// TIA Portal V18 export
FUNCTION "TCS" : Void   // FC3, LAD
{ S7_Optimized_Access := 'TRUE' }
VERSION : 0.1
// stored: AutoNumber true, IsIECCheckEnabled false, SetENOAutomatically false, UDAEnableTagReadback false
BEGIN

REGION Network 1
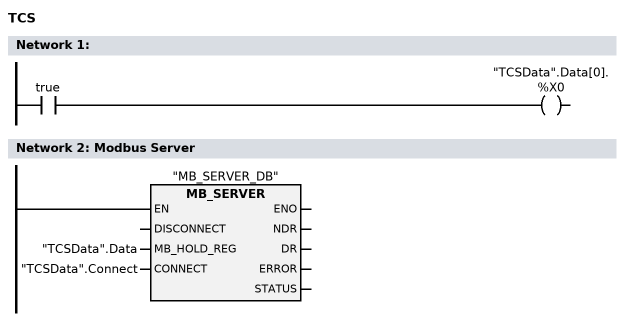
   RUNG wire#powerrail
      Contact( true )
      Coil( "TCSData".Data[0].%X0 )
   END_RUNG
   // the same network as SCL:
   "TCSData".Data[0].%X0 := true;
END_REGION

REGION Network 2: Modbus Server
   RUNG wire#powerrail
      "MB_SERVER_DB".MB_SERVER(DISCONNECT :=, MB_HOLD_REG := "TCSData".Data, CONNECT := "TCSData".Connect, NDR =>, DR =>, ERROR =>, STATUS =>)
   END_RUNG
   // the same network as SCL:
   "MB_SERVER_DB"(MB_HOLD_REG := "TCSData".Data, CONNECT := "TCSData".Connect);   // MB_SERVER
END_REGION
END_FUNCTION
